PROGRAM MAIN
VAR
END_VAR

END_PROGRAM

(* stored: Version 1.1.0.1
   POU MAIN: Id {e030a0ad-d647-47b9-9185-933745c41f93} *)
